FUNCTION_BLOCK MotorDegreeToCablePosition
VAR_IN_OUT
	motor_position : LREAL;	// deg/s
	reset_cable_position : BOOL;	
END_VAR
VAR_OUTPUT
	cable_position : LREAL;
END_VAR
VAR
	winch_radius : LREAL := 16.0;
END_VAR
VAR PERSISTENT
	motor_position_shift : LREAL;
END_VAR

IF reset_cable_position THEN
	motor_position_shift := motor_position;
END_IF

cable_position := (motor_position - motor_position_shift) * Tc2_System.PI / 180.0 * winch_radius;

END_FUNCTION_BLOCK

(* stored: Version 1.1.0.1, ProductVersion 3.1.4024.11
   POU MotorDegreeToCablePosition: Id {f08e5447-b4e4-47a6-9e6f-4eca85de6f25}, SpecialFunc None *)
